// TIA Portal V20 export
VAR_GLOBAL   // PLC tag table "SSP2"
   SSP2_Valve_Up AT %Q5201.0 : Bool;
   SSP2_Valve_Down AT %Q5201.1 : Bool;
   SSP2_Hydraulic_Unit AT %Q5201.2 : Bool;
   SSP2_Sen_Drv_1 AT %I5202.0 : Bool;
   SSP2_Sen_Drv_2 AT %I5202.1 : Bool;
   SSP2_Sen_Drv_3 AT %I5202.2 : Bool;
   SSP2_Sen_Drv_4 AT %I5202.3 : Bool;
   SSP2_Sen_Val1_Up AT %I5202.4 : Bool;
   SSP2_Sen_Val1_Down AT %I5202.5 : Bool;
   SSP2_Sen_Val2_Up AT %I5202.6 : Bool;
   SSP2_Sen_Val2_Down AT %I5202.7 : Bool;
   SSP2_Hyd_Filtr AT %I5203.0 : Bool;
   SSP2_Hyd_Empty AT %I5203.1 : Bool;
   SSP2_Safety1_1 AT %I5273.0 : Bool;
   SSP2_Safety2_1 AT %I5273.1 : Bool;
   SSP2_Safety3_1 AT %I5273.2 : Bool;
   SSP2_Safety4_1 AT %I5273.3 : Bool;
   SSP2_Safety1_2 AT %I5274.0 : Bool;
   SSP2_Safety2_2 AT %I5274.1 : Bool;
   SSP2_Safety3_2 AT %I5274.2 : Bool;
   SSP2_Safety4_2 AT %I5274.3 : Bool;
END_VAR
